{attribute 'GeneratedUsingTerminal: EL6080-0000-0018'}
{attribute addProperty BoxType "EL6080-0000-0018"}
{attribute addProperty Description "EL6080 EtherCAT Memory Terminal (128kB)"}
{attribute addProperty Physics "KK"}
{attribute addProperty Id "StatusAT %I*Status_07D3AAF62InputsEMPTY_STRUCTURE0ControlAT %Q*Control_DAFD38E02OutputsEMPTY_STRUCTURE0WcStateAT %I*WcState_9091E0EB2InfoDataAT %I*InfoData_32EB74EA10"}
{attribute addProperty CRC "2640427583"}
{attribute addProperty Size "16"}
TYPE EL6080_9D61BA3F EXTENDS EtcSlaveTerminalBase_947E5A46 :
STRUCT
	{attribute addProperty Name "Status"}
	Status : Status_07D3AAF6;
	{attribute addProperty Name "Inputs"}
	Inputs : EMPTY_STRUCTURE;
	{attribute addProperty Name "Control"}
	Control : Control_DAFD38E0;
	{attribute addProperty Name "Outputs"}
	Outputs : EMPTY_STRUCTURE;
	{attribute addProperty Name "WcState"}
	WcState : WcState_9091E0EB;
	{attribute addProperty Name "InfoData"}
	InfoData : InfoData_32EB74EA;
END_STRUCT
END_TYPE

(* stored: Version 1.2.0.0, ProductVersion 3.1.4024.11
   DUT EL6080_9D61BA3F: Id {9d44c0a3-8fe2-4a46-9c2c-a832116ae98b} *)
